// Mitsubishi GX Works2 project: LADDER_code   PLC: FX3U/FX3UC

PROGRAM MAIN
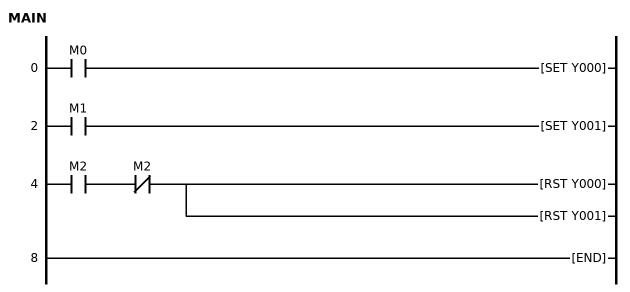
0     LD      M0
      SET     Y000
2     LD      M1
      SET     Y001
4     LD      M2
      ANI     M2
      RST     Y000
      RST     Y001
8     END
END_PROGRAM
